FUNCTION_BLOCK Test_F_DateTimeAsString_ms_ReturnsDateTimeString EXTENDS TUnitTestBase
VAR
    TimeStruct : TIMESTRUCT := (wDay := 23, wMonth := 12, wYear := 1945, wHour := 22, wMinute := 20, wSecond := 18, wMilliseconds := 512);
END_VAR

Assertion.AssertEquals_STRING(
    Expected := '22:20:18.512 23/12/1945',
    Actual   := F_DateTimeAsString_ms(TimeStruct),
    ObjectName := _TestName,
    VariableName  := 'F_DateTimeAsString_ms(TimeStruct)');


TestFinished();

END_FUNCTION_BLOCK

(* stored: Version 1.1.0.1, ProductVersion 3.1.4024.4
   POU Test_F_DateTimeAsString_ms_ReturnsDateTimeString: Id {3b9edf74-0e2a-0b80-276d-9d87de77dccc}, SpecialFunc None *)
